// TIA Portal project "Practica_5" (V14)
// Automatización de una planta de envasado de pelotitas.

(* hardware
DEVICE "S7-1200 station_1"  S7-1200 Station
   slot 0: "Rack_0"  S7-1200 Rack  Rack  V1.0
   slot 1: "PLC_1"  CPU 1214C DC/DC/DC  6ES7 214-1AG40-0XB0  V4.2
*)

// ===== PLC "PLC_1"  CPU 1214C DC/DC/DC =====

VAR_GLOBAL   // PLC tag table "Default tag table"
   "Q_P2" AT %Q0.1 : Bool;
   "I_PM" AT %I0.0 : Bool;
   "I_PP" AT %I0.1 : Bool;
   "Q_P1" AT %Q0.0 : Bool;
END_VAR

DATA_BLOCK "PUT_ALTERNATED_BALLS_DB"   // DB1
{ S7_Optimized_Access := 'TRUE' }
VERSION : 0.1
// stored: InstanceOfName PUT_ALTERNATED_BALLS
"PUT_ALTERNATED_BALLS"
BEGIN
END_DATA_BLOCK

FUNCTION_BLOCK "PUT_ALTERNATED_BALLS"   // FB1, LAD
{ S7_Optimized_Access := 'TRUE' }
VERSION : 0.1
   VAR_INPUT
      PM : Bool := false;
      PP : Bool := false;
   END_VAR
   VAR_OUTPUT
      ACCIONAR_P1 : Bool;
      ACCIONAR_P2 : Bool;
   END_VAR
   VAR
      ENCENDIDO : Bool;
      APAGADO : Bool;
      MEMORIA_P : Bool;
   END_VAR
   VAR RETAIN
      CONTADOR_BOLITAS : CTU_INT;
      ACCIONAR_P2_ST : Bool;
      ACCIONAR_P1_ST : Bool;
   END_VAR
   VAR
      TIMER_TON_P2 : TON_TIME;
      MEMORIA_PM : Bool;
      TIMER_TOF_P2 : TOF_TIME;
   END_VAR
   VAR CONSTANT
      TIEMPO_ACCIONAR_P1 : Time := T#2s;
      TIEMPO_ACCIONAR_P2 : Time := T#2s;
      PARES_DE_BOLITAS : Int := 5;
   END_VAR
   VAR_TEMP   // added for the SCL form of the ladder/FBD networks
      _w1 : Bool;
   END_VAR
BEGIN

REGION Network 1
   // Inicialización
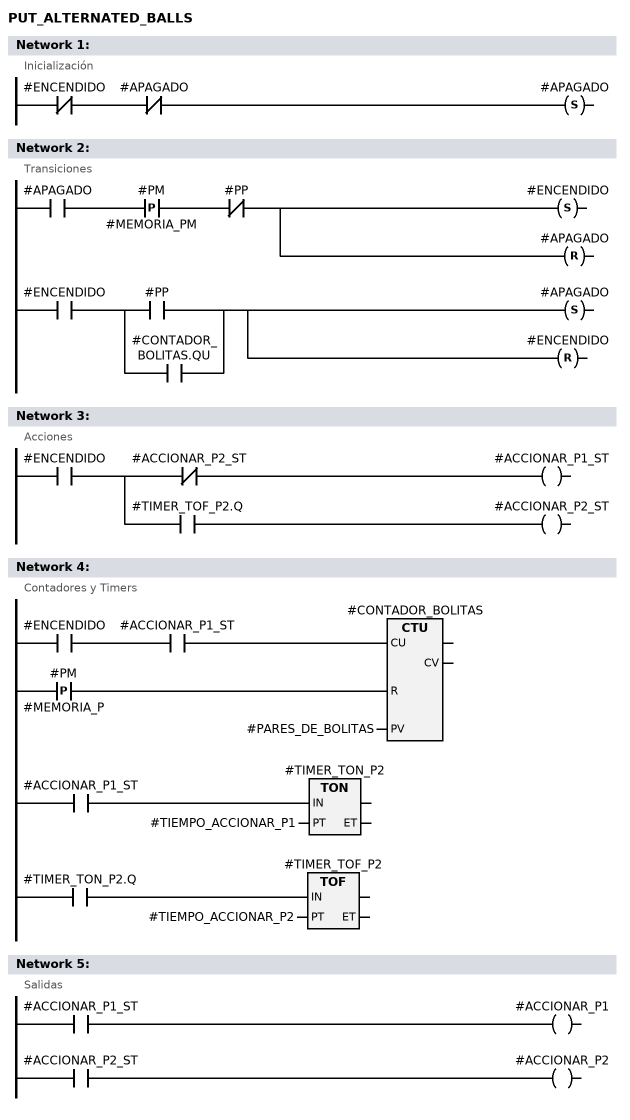
   RUNG wire#powerrail
      I_Contact( #ENCENDIDO )
      I_Contact( #APAGADO )
      S_Coil( #APAGADO )
   END_RUNG
   // the same network as SCL:
   IF NOT #ENCENDIDO AND NOT #APAGADO THEN #APAGADO := TRUE; END_IF;
END_REGION

REGION Network 2
   // Transiciones
   RUNG wire#powerrail
      Contact( #APAGADO )
      P_Contact(operand := #PM, bit := #MEMORIA_PM)
      I_Contact( #PP )
      wire#w1
      S_Coil( #ENCENDIDO )
   END_RUNG
   RUNG wire#w1
      R_Coil( #APAGADO )
   END_RUNG
   RUNG wire#powerrail
      Contact( #ENCENDIDO )
      wire#w2
      Contact( #PP )
      wire#w3
      S_Coil( #APAGADO )
   END_RUNG
   RUNG wire#w2
      Contact( #CONTADOR_BOLITAS.QU )
   END_RUNG wire#w3
   RUNG wire#w3
      R_Coil( #ENCENDIDO )
   END_RUNG
   // the same network as SCL:
   #_w1 := #APAGADO AND #PM AND NOT #MEMORIA_PM;   // rising edge of #PM
   #MEMORIA_PM := #PM;
   IF #_w1 AND NOT #PP THEN
       #ENCENDIDO := TRUE;
       #APAGADO := FALSE;
   END_IF;
   IF #ENCENDIDO AND (#PP OR #CONTADOR_BOLITAS.QU) THEN
       #APAGADO := TRUE;
       #ENCENDIDO := FALSE;
   END_IF;
END_REGION

REGION Network 3
   // Acciones
   RUNG wire#powerrail
      Contact( #ENCENDIDO )
      wire#w1
      I_Contact( #ACCIONAR_P2_ST )
      Coil( #ACCIONAR_P1_ST )
   END_RUNG
   RUNG wire#w1
      Contact( #TIMER_TOF_P2.Q )
      Coil( #ACCIONAR_P2_ST )
   END_RUNG
   // the same network as SCL:
   #ACCIONAR_P1_ST := #ENCENDIDO AND NOT #ACCIONAR_P2_ST;
   #ACCIONAR_P2_ST := #ENCENDIDO AND #TIMER_TOF_P2.Q;
END_REGION

REGION Network 4
   // Contadores y Timers
   #_w1 := #PM AND NOT #MEMORIA_P;   // rising edge of #PM
   #MEMORIA_P := #PM;
   #CONTADOR_BOLITAS(CU := #ENCENDIDO AND #ACCIONAR_P1_ST, R := #_w1, PV := #PARES_DE_BOLITAS);   // CTU
   #TIMER_TON_P2(IN := #ACCIONAR_P1_ST, PT := #TIEMPO_ACCIONAR_P1);   // TON
   #TIMER_TOF_P2(IN := #TIMER_TON_P2.Q, PT := #TIEMPO_ACCIONAR_P2);   // TOF
END_REGION

REGION Network 5
   // Salidas
   RUNG wire#powerrail
      Contact( #ACCIONAR_P1_ST )
      Coil( #ACCIONAR_P1 )
   END_RUNG
   RUNG wire#powerrail
      Contact( #ACCIONAR_P2_ST )
      Coil( #ACCIONAR_P2 )
   END_RUNG
   // the same network as SCL:
   #ACCIONAR_P1 := #ACCIONAR_P1_ST;
   #ACCIONAR_P2 := #ACCIONAR_P2_ST;
END_REGION
END_FUNCTION_BLOCK

ORGANIZATION_BLOCK "Main"   // OB1, LAD, ProgramCycle
TITLE = "Main Program Sweep (Cycle)"
{ S7_Optimized_Access := 'TRUE' }
VERSION : 0.1
   VAR_INPUT
      Initial_Call : Bool;   // Initial call of this OB
      Remanence : Bool;   // =True, if remanent data are available
   END_VAR
BEGIN

REGION Network 1
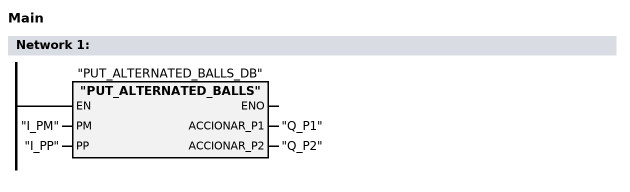
   RUNG wire#powerrail
      "PUT_ALTERNATED_BALLS_DB"(PM := "I_PM", PP := "I_PP", ACCIONAR_P1 => "Q_P1", ACCIONAR_P2 => "Q_P2")
   END_RUNG
   // the same network as SCL:
   "PUT_ALTERNATED_BALLS_DB"(PM := "I_PM", PP := "I_PP", ACCIONAR_P1 => "Q_P1", ACCIONAR_P2 => "Q_P2");   // "PUT_ALTERNATED_BALLS"
END_REGION
END_ORGANIZATION_BLOCK